FUNCTION Update_Jobe_State : BOOL
VAR_INPUT
	Camera : REFERENCE TO Cognex_Camera;
END_VAR
VAR
END_VAR

IF NOT Camera.CameraState = Camera_State.Jope_Running THEN
	RETURN;
END_IF

IF Camera.JobeState = Job_State.TriggerAck THEN
	IF Camera.AcquisitionStatusRegister.Acquistion_Trigger_Acknowledge THEN
		Camera.JobeState := Job_State.Wate;
		Camera.AcquisitionControl.Clear_Exposure_Complete := FALSE;
		Camera.AcquisitionControl.Acquistion_Trigger := FALSE;
		RETURN;
	ELSE
		RETURN;
	END_IF
ELSIF Camera.JobeState = Job_State.Wate THEN
	IF Camera.InspectionStatusRegister.Inspection_Completed AND (NOT Camera.InspectionStatusRegister.System_Busy) THEN
		Camera.JobeState := Job_State.Complte;
	END_IF
	
ELSIF Camera.InspectionStatusRegister.Error THEN
	Camera.JobeState := Job_State.Error;
	Camera.CameraState := Camera_State.Error;
	CASE Camera.ErrorCode OF
		16#0100: // Trigger set while disabeld
			Camera.Error := Camera_Error.Trigger_Set_While_disabeld;
		16#0101: // trigger set while offline
			Camera.Error := Camera_Error.Trigger_Set_While_Offline;
		16#0400: // already executing error
			Camera.Error := Camera_Error.Already_Executing;
		16#0401: // job load requeted while online
			Camera.Error := Camera_Error.Job_Load_Requested_While_Online;
		16#0402: // job load requested does not exist on the camera
			Camera.Error := Camera_Error.Job_Does_Not_Exist;
	END_CASE
ELSIF Camera.JobeState = Job_State.Error THEN
	RETURN;
ELSE
	Camera.JobeState := Job_State.Error;
	Camera.Error := Camera_Error.StateError;
	RETURN;
END_IF

END_FUNCTION

(* stored: Version 1.1.0.1, ProductVersion 3.1.4024.10
   POU Update_Jobe_State: Id {1b98cabf-e7a1-488d-8010-b77c8a056498}, SpecialFunc None *)
